FUNCTION TryConvert_LWORD_TO_TIME : BOOL
VAR_INPUT
	in : LWORD;
	out : REFERENCE TO TIME;
END_VAR

IF in > DatatypeLimits.MAX_VALUE_OF_LWORD_WHICH_CAN_BE_HELD_IN_A_TIME THEN
	RETURN;
END_IF

out := LWORD_TO_TIME(in);
TryConvert_LWORD_TO_TIME := TRUE;

END_FUNCTION

(* stored: Version 1.1.0.1, ProductVersion 3.1.4024.12
   POU TryConvert_LWORD_TO_TIME: Id {2f2fa885-ff62-456a-8f1a-f4e885f4ebca}, SpecialFunc None *)
